# EPICS substitutions: epics/support/quadEM-R9-2-1/iocBoot/iocNSLS2_EM/DACs.substitutions
file "$(QUADEM)/db/NSLS2_DAC.template"
{
pattern
{P,               R,     N, PORT,     EGUL,   DRVL,  LOPR,  EGUF,  DRVH,   HOPR, PREC,  LINR}
{quadEMTest:, NSLS2_EM:, 0, NSLS2_EM,  -10,   -10,   -10,    10,   10.,    10.,  4,     LINEAR}
{quadEMTest:, NSLS2_EM:, 1, NSLS2_EM,  -10,   -10,   -10,    10,   10.,    10.,  4,     LINEAR}
{quadEMTest:, NSLS2_EM:, 2, NSLS2_EM,  -10,   -10,   -10,    10,   10.,    10.,  4,     LINEAR}
{quadEMTest:, NSLS2_EM:, 3, NSLS2_EM,  -10,   -10,   -10,    10,   10.,    10.,  4,     LINEAR}
}
